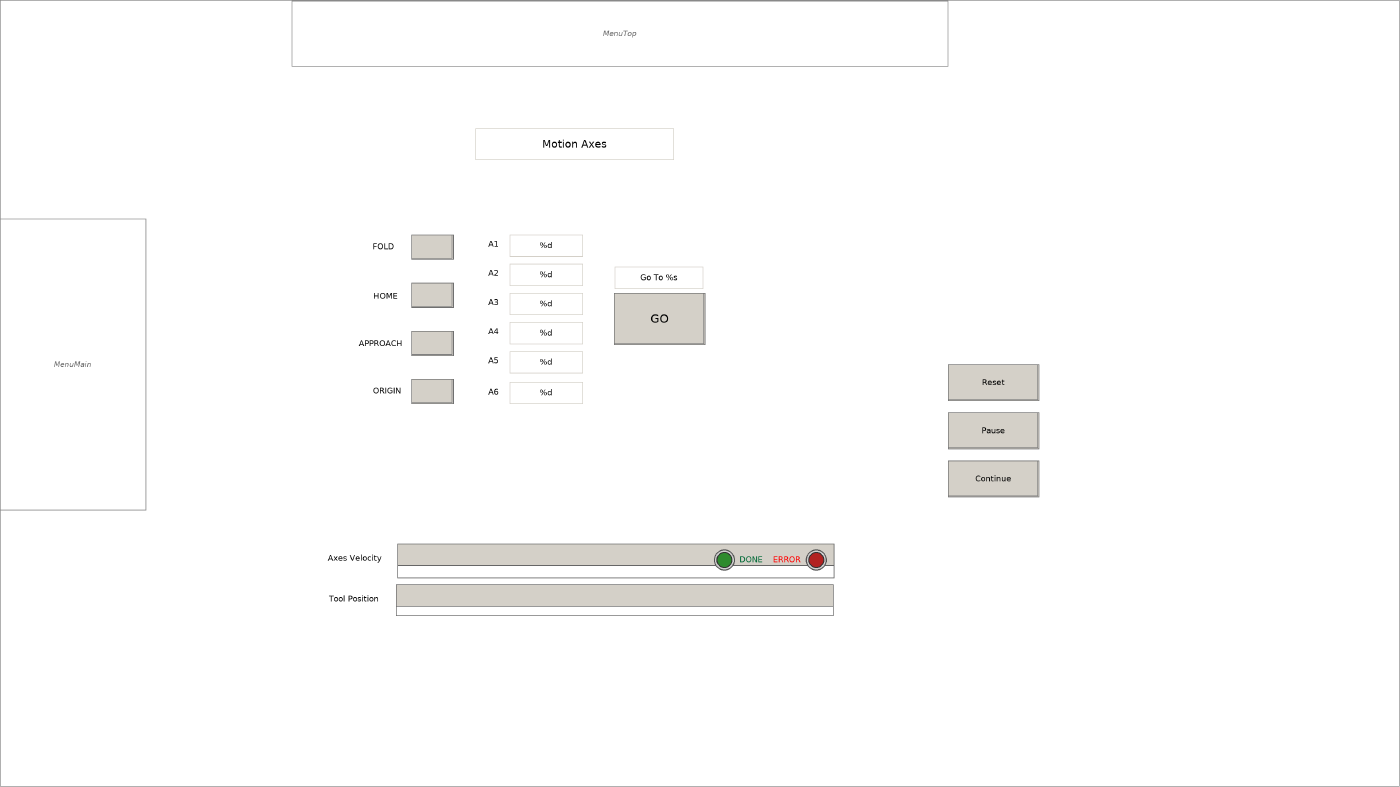
VISUALIZATION Motion_Axes  // 1920x1080
    Frame (400,1 900x90)
        shows MenuTop()
    Frame (0,300 200x400)
        shows MenuMain()
    Textfield (652,176 272x43), "Motion Axes"
    Button (1300,566 125x50), "Pause"
        tap mxA_Motion.fbAutoDemo.fbKRC_Interrupt.Execute
    Button (1300,632 125x50), "Continue"
        tap mxA_Motion.fbAutoDemo.fbKRC_Continue.Enable
    Button (842,402 125x71), "GO"
        tap MAIN.Move_Axes.Execute
    Textfield (699,322 100x30), "%d", text variable: MAIN.Move_Axes.AxisPosition.A1
    Textfield (699,362 100x30), "%d", text variable: MAIN.Move_Axes.AxisPosition.A2
    Textfield (699,402 100x30), "%d", text variable: MAIN.Move_Axes.AxisPosition.A3
    Textfield (699,442 100x30), "%d", text variable: MAIN.Move_Axes.AxisPosition.A4
    Textfield (699,482 100x30), "%d", text variable: MAIN.Move_Axes.AxisPosition.A5
    Textfield (699,524 100x30), "%d", text variable: MAIN.Move_Axes.AxisPosition.A6
    Label (660,323 34x24), "A1"
    Label (660,363 34x24), "A2"
    Label (660,403 34x24), "A3"
    Label (660,443 34x24), "A4"
    Label (660,483 34x24), "A5"
    Label (660,526 34x24), "A6"
    Button (1300,500 125x50), "Reset"
        tap MAIN.Write_Program_Abort.ExecuteCmd
    Label (506,392 46x29), "HOME"
    Label (505,324 42x29), "FOLD"
    Label (487,457 70x29), "APPROACH"
    Label (508,522 46x29), "ORIGIN"
    Button (564,322 58x34)
        OnMouseDown: execute {
            main.Move_Axes.AxisPosition.A1:=-90;
            main.Move_Axes.AxisPosition.A2:=-108;
            main.Move_Axes.AxisPosition.A3:=110;
            main.Move_Axes.AxisPosition.A4:=1;
            main.Move_Axes.AxisPosition.A5:=25;
            main.Move_Axes.AxisPosition.A6:=1;
            gvl_gui.GlobalPositionString := TO_STRING("FOLD");
        }
    Button (564,388 58x34)
        OnMouseClick: execute {
            main.Move_Axes.AxisPosition.A1:=-66;
            main.Move_Axes.AxisPosition.A2:=-90;
            main.Move_Axes.AxisPosition.A3:=70;
            main.Move_Axes.AxisPosition.A4:=1;
            main.Move_Axes.AxisPosition.A5:=15;
            main.Move_Axes.AxisPosition.A6:=1;
            gvl_gui.GlobalPositionString := TO_STRING("Home");
        }
    Button (564,454 58x34)
        OnMouseClick: execute {
            main.Move_Axes.AxisPosition.A1:=1;
            main.Move_Axes.AxisPosition.A2:=-100;
            main.Move_Axes.AxisPosition.A3:=60;
            main.Move_Axes.AxisPosition.A4:=1;
            main.Move_Axes.AxisPosition.A5:=40;
            main.Move_Axes.AxisPosition.A6:=1;
            gvl_gui.GlobalPositionString := TO_STRING("Approach");
        }
    Button (564,520 58x34)
        OnMouseClick: execute {
            main.Move_Axes.AxisPosition.A1:=1;
            main.Move_Axes.AxisPosition.A2:=-70;
            main.Move_Axes.AxisPosition.A3:=50;
            main.Move_Axes.AxisPosition.A4:=1;
            main.Move_Axes.AxisPosition.A5:=20;
            main.Move_Axes.AxisPosition.A6:=1;
            gvl_gui.GlobalPositionString := TO_STRING("Origin");
        }
    Textfield (843,366 121x30), "Go To %s", text variable: GVL_GUI.GlobalPositionString
    Table (543,802 600x43), data array: mxA_Motion.fbKRC_ReadActualPosition.Position
        p3854506369: mxA_Motion.fbKRC_ReadActualPosition.Position.X
        p1892666644: mxA_Motion.fbKRC_ReadActualPosition.Position.Y
        p338671338: mxA_Motion.fbKRC_ReadActualPosition.Position.Z
        p2170511999: mxA_Motion.fbKRC_ReadActualPosition.Position.A
        p3723444502: mxA_Motion.fbKRC_ReadActualPosition.Position.B
        p1218418051: mxA_Motion.fbKRC_ReadActualPosition.Position.C
        p746581629: mxA_Motion.fbKRC_ReadActualPosition.Position.Status
        p3104783080: mxA_Motion.fbKRC_ReadActualPosition.Position.Turn
        p2501879983: mxA_Motion.fbKRC_ReadActualPosition.Position.E1
        p7306298: mxA_Motion.fbKRC_ReadActualPosition.Position.E2
        p1933151965: mxA_Motion.fbKRC_ReadActualPosition.Position.E3
        p3863566920: mxA_Motion.fbKRC_ReadActualPosition.Position.E4
        p2192122294: mxA_Motion.fbKRC_ReadActualPosition.Position.E5
        p400160035: mxA_Motion.fbKRC_ReadActualPosition.Position.E6
        p1757482276: status
        p4088588272: turn
    Table (545,746 599x47), data array: Read_Axes_Velocity.ReadAxesVelocity
        p3854506369: Read_Axes_Velocity.ReadAxesVelocity.AxisGroupIdx
        p1892666644: Read_Axes_Velocity.ReadAxesVelocity.ExecuteCmd
        p338671338: Read_Axes_Velocity.ReadAxesVelocity.Done
        p2170511999: Read_Axes_Velocity.ReadAxesVelocity.Error
        p3723444502: Read_Axes_Velocity.ReadAxesVelocity.ErrorID
        p1218418051: Read_Axes_Velocity.ReadAxesVelocity.A1
        p746581629: Read_Axes_Velocity.ReadAxesVelocity.A2
        p3104783080: Read_Axes_Velocity.ReadAxesVelocity.A3
        p2501879983: Read_Axes_Velocity.ReadAxesVelocity.A4
        p7306298: Read_Axes_Velocity.ReadAxesVelocity.A5
        p1933151965: Read_Axes_Velocity.ReadAxesVelocity.A6
        p3863566920: Read_Axes_Velocity.ReadAxesVelocity.E1
        p2192122294: Read_Axes_Velocity.ReadAxesVelocity.E2
        p400160035: Read_Axes_Velocity.ReadAxesVelocity.E3
        p1265227338: Read_Axes_Velocity.ReadAxesVelocity.E4
        p3726181087: Read_Axes_Velocity.ReadAxesVelocity.E5
        p3136911649: Read_Axes_Velocity.ReadAxesVelocity.E6
        p797552052: Read_Axes_Velocity.ReadAxesVelocity.mxA_ExecuteCommand
    Rectangle (440,751 93x30), "Axes Velocity"
    Lamp1 (977,752 33x33), variable: Read_Axes_Velocity.ReadAxesVelocity.Done, style: Lamp-Lamp1-Green
    Lamp1 (1103,752 33x33), variable: Read_Axes_Velocity.ReadAxesVelocity.Error, style: Lamp-Lamp1-Red
    Rectangle (1007,757 46x22), "DONE"
    Rectangle (1056,757 46x22), "ERROR"
    Rectangle (439,807 93x30), "Tool Position"
END_VISUALIZATION

(* stored: Version 1.1.0.1, ProductVersion 3.1.4024.10
   Visu Motion_Axes: Id {fa9dda43-7992-4a47-a4bc-3e3fd0c6c535} *)
